// Writes an uint32 field value, without a tag, to the stream.
FUNCTION F_WriteUInt32 : HRESULT
VAR_IN_OUT      
    stCtx : ST_WriteContext;
END_VAR
VAR_INPUT
    nValue : UDINT;
END_VAR
VAR
END_VAR


F_WriteUInt32 := F_WriteRawVarint32(stCtx, nValue);

END_FUNCTION

(* stored: Version 1.1.0.1
   POU F_WriteUInt32: Id {e04e4398-e727-4746-9f66-4ec11446c061}, SpecialFunc None *)
